Staubli VAL3: exceptionRos.pgx

public program exceptionRos(FlagStatus& x_fRosStatus, num& x_nRosFlagCmd)
begin

  //This program is used for checking the ROS command of exception handling from the host ROS controller
  //and deciding whether the robot should keep executing the motion command or not.

  //The ROS command flag from the host ROS controller should be acquired through TCP/IP socket communication.
  //And the ROS flag in the ROS massage command is in the last element in the received array.
  x_fRosStatus.RosFlag=x_nRosFlagCmd

end
